FUNCTION_BLOCK DEV_Valve EXTENDS FB_DeviceBase IMPLEMENTS ITF_Valve

VAR
	I_FeedbackOpen		AT	%I* : BOOL;
	I_FeedbackClosed 	AT 	%I* : BOOL;
	I_Estop				AT	%I*	: BOOL;
	Q_ValveOutput		AT	%Q*	: BOOL;
	
	s_eActualState				: E_ValveState;
	s_eOperatingMode			: E_OperationMode;
	s_tonFeedbackTime			: TON;
	
	bFeedbackError		: BOOL;
	bEstopActive		: BOOL;
	bBothFeedback		: BOOL;
END_VAR

METHOD _FExceptions : BOOL
VAR_INPUT
END_VAR
END_METHOD

METHOD PRIVATE _StHmi
VAR_INPUT
	stHMI : stDevValve;
END_VAR
END_METHOD

{warning 'add property implementation'}
PROPERTY ActualState : E_ValveState
GET
END_GET
END_PROPERTY

{warning 'add method implementation '}
METHOD Close : BOOL
END_METHOD

{warning 'add property implementation'}
PROPERTY EmergencyStatus : BOOL
GET
END_GET
END_PROPERTY

{warning 'add method implementation '}
METHOD Open : BOOL
END_METHOD

{warning 'add property implementation'}
PROPERTY OperatingMode : BOOL
GET
END_GET
END_PROPERTY

{warning 'add method implementation '}
METHOD Reset : BOOL
END_METHOD

{warning 'add method implementation '}
METHOD SetMode : BOOL
END_METHOD

END_FUNCTION_BLOCK

(* stored: Version 1.1.0.1, ProductVersion 3.1.4024.12
   POU DEV_Valve: Id {36449132-d53d-484c-9ebb-e20c5d923732}, SpecialFunc None
   Folder Method: Id {e939ec98-8b7a-4b1e-af4c-b16997f2a20a}
   Folder Properties: Id {e5ddc51b-0b4a-4524-a37b-63772754452c}
   Method _FExceptions: Id {4182cdba-02cc-4eab-a4ed-e50d2a21d2b2}
   Method _StHmi: Id {4857c0f1-bb49-4ade-a221-03c3da4527f3}
   Property ActualState: Id {931ebd17-2b5f-4423-8f65-7ddf693cfc54}
   Get Get: Id {d15455c8-edf5-4df5-93b3-199038b24bd6}
   Method Close: Id {aca272f9-81f8-4175-862d-610a22b53210}
   Property EmergencyStatus: Id {faebb791-9d9b-43b6-a8d9-17b06181c36a}
   Get Get: Id {c3cce2a6-d6bf-4e0b-85f6-735f99dda6a1}
   Method Open: Id {0dd4219c-86e8-4ce9-a367-53dcd4f1bc91}
   Property OperatingMode: Id {7a40270e-1e41-448a-af48-293399f4e85d}
   Get Get: Id {ed17de1b-e5c2-4d93-978b-ef4e92e8ae6c}
   Method Reset: Id {17aa9f20-5165-42a4-9d4c-661c80698cc6}
   Method SetMode: Id {dae04c1b-0e2a-44f9-aed5-12adf790a98c} *)
